// TIA Portal V19 export
FUNCTION "FinalCutLub_CALL" : Void   // FC169, LAD
TITLE = PRESS TOOLS LUBRICATION
// stored: SetENOAutomatically false
BEGIN

REGION Network 1: Data In (Pb)
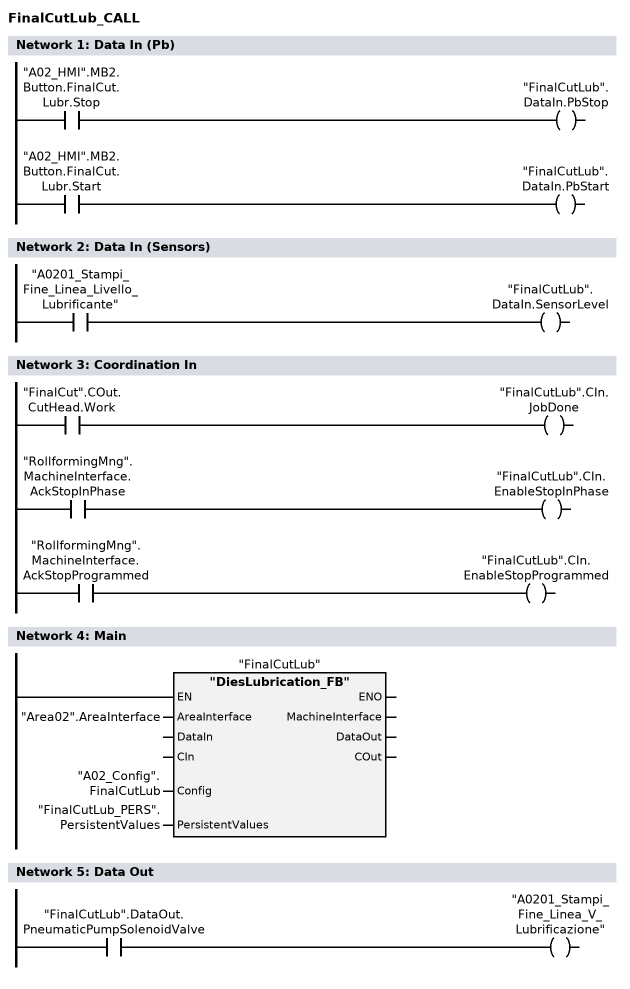
   RUNG wire#powerrail
      Contact( "A02_HMI".MB2.Button.FinalCut.Lubr.Stop )
      Coil( "FinalCutLub".DataIn.PbStop )
   END_RUNG
   RUNG wire#powerrail
      Contact( "A02_HMI".MB2.Button.FinalCut.Lubr.Start )
      Coil( "FinalCutLub".DataIn.PbStart )
   END_RUNG
   // the same network as SCL:
   "FinalCutLub".DataIn.PbStop := "A02_HMI".MB2.Button.FinalCut.Lubr.Stop;
   "FinalCutLub".DataIn.PbStart := "A02_HMI".MB2.Button.FinalCut.Lubr.Start;
END_REGION

REGION Network 2: Data In (Sensors)
   RUNG wire#powerrail
      Contact( "A0201_Stampi_Fine_Linea_Livello_Lubrificante" )
      Coil( "FinalCutLub".DataIn.SensorLevel )
   END_RUNG
   // the same network as SCL:
   "FinalCutLub".DataIn.SensorLevel := "A0201_Stampi_Fine_Linea_Livello_Lubrificante";
END_REGION

REGION Network 3: Coordination In
   RUNG wire#powerrail
      Contact( "FinalCut".COut.CutHead.Work )
      Coil( "FinalCutLub".CIn.JobDone )
   END_RUNG
   RUNG wire#powerrail
      Contact( "RollformingMng".MachineInterface.AckStopInPhase )
      Coil( "FinalCutLub".CIn.EnableStopInPhase )
   END_RUNG
   RUNG wire#powerrail
      Contact( "RollformingMng".MachineInterface.AckStopProgrammed )
      Coil( "FinalCutLub".CIn.EnableStopProgrammed )
   END_RUNG
   // the same network as SCL:
   "FinalCutLub".CIn.JobDone := "FinalCut".COut.CutHead.Work;
   "FinalCutLub".CIn.EnableStopInPhase := "RollformingMng".MachineInterface.AckStopInPhase;
   "FinalCutLub".CIn.EnableStopProgrammed := "RollformingMng".MachineInterface.AckStopProgrammed;
END_REGION

REGION Network 4: Main
   RUNG wire#powerrail
      "FinalCutLub"(AreaInterface := "Area02".AreaInterface, DataIn :=, CIn :=, Config := "A02_Config".FinalCutLub, PersistentValues := "FinalCutLub_PERS".PersistentValues, MachineInterface =>, DataOut =>, COut =>)
   END_RUNG
   // the same network as SCL:
   "FinalCutLub"(AreaInterface := "Area02".AreaInterface,   // "DiesLubrication_FB"
                 Config := "A02_Config".FinalCutLub,
                 PersistentValues := "FinalCutLub_PERS".PersistentValues);
END_REGION

REGION Network 5: Data Out
   RUNG wire#powerrail
      Contact( "FinalCutLub".DataOut.PneumaticPumpSolenoidValve )
      Coil( "A0201_Stampi_Fine_Linea_V_Lubrificazione" )
   END_RUNG
   // the same network as SCL:
   "A0201_Stampi_Fine_Linea_V_Lubrificazione" := "FinalCutLub".DataOut.PneumaticPumpSolenoidValve;
END_REGION
END_FUNCTION
